FUNCTION_BLOCK FB_ParseString
VAR_INPUT
	sCharToSearch : STRING;
	sInputString  : STRING;
END_VAR
VAR_OUTPUT
	sStringParsed : STRING;
END_VAR
VAR
	Position: INT;
END_VAR

Position := FIND(sInputString, sCharToSearch);
sStringParsed := DELETE(sInputString, Position, LEN(sInputString));

END_FUNCTION_BLOCK

(* stored: Version 1.1.0.1, ProductVersion 3.1.4024.12
   POU FB_ParseString: Id {7d98a99a-5b8c-4463-bed0-a0efa1e6537d}, SpecialFunc None *)
